FUNCTION F_EnsureMaxVelo: BOOL
VAR_IN_OUT
	fNextVeloX : LREAL;
	fNextVeloY : LREAL;
END_VAR
VAR
	fNormNextVelo : LREAL;
	fNextVeloUnitLength : LREAL;
END_VAR

fNormNextVelo := TO_LREAL(F_2Norm(fA := TO_REAL(fNextVeloX), fB := TO_REAL(fNextVeloY)));
IF fNormNextVelo > GVL.fMaxVelo THEN
	fNextVeloX := (fNextVeloX/fNormNextVelo) * GVL.fMaxVelo;
	fNextVeloY := (fNextVeloY/fNormNextVelo) * GVL.fMaxVelo;
	F_EnsureMaxVelo := TRUE;
END_IF
F_EnsureMaxVelo := FALSE;

END_FUNCTION

(* stored: Version 1.1.0.1, ProductVersion 3.1.4024.12
   POU F_EnsureMaxVelo: Id {16893116-0d2a-4350-9d82-f09f1a19198a}, SpecialFunc None *)
